(* IEC 61131-3 sources: eCockpitGit/test_project/src/%F%00 Library/%F%Common Functions/%F%Bits/%F%Bit Get Part, 8 files *)

(* ---- %POU%FU_bBitGetPart.st ---- *)
//This function gets only the needed bits of a variable
// |**Version**|**Author**| **Date** |**Changes**
// | 1         | NSN      | 16-03-22 | Creation
FUNCTION FU_bBitGetPart : BYTE
VAR_INPUT
	value			:BYTE;		//Variable to get value from
	amount			:BYTE;		//Amount of bits to change
	offset			:BYTE;		//Offset in variable to change bits at
END_VAR
(*%!%__DELIMITER__%!%*)
FU_bBitPartThrough		:=		SHR(value,offset) AND GConstants.binaryMaskByte[amount];

(* ---- %POU%FU_diBitGetPart.st ---- *)
//This function gets only the needed bits of a variable
// |**Version**|**Author**| **Date** |**Changes**
// | 1         | NSN      | 16-03-22 | Creation
FUNCTION FU_diBitGetPart : DINT
VAR_INPUT
	value			:DINT;		//Variable to get value from
	amount			:BYTE;		//Amount of bits to change
	offset			:BYTE;		//Offset in variable to change bits at
END_VAR
(*%!%__DELIMITER__%!%*)
FU_diBitGetPart		:=		TO_DINT(TO_UDINT(SHR(value,offset)) AND TO_UDINT(GConstants.binaryMaskDint[amount]));

(* ---- %POU%FU_dwBitGetPart.st ---- *)
//This function gets only the needed bits of a variable
// |**Version**|**Author**| **Date** |**Changes**
// | 1         | NSN      | 16-03-22 | Creation
FUNCTION FU_dwBitGetPart : DWORD
VAR_INPUT
	value			:DWORD;		//Variable to get value from
	amount			:BYTE;		//Amount of bits to change
	offset			:BYTE;		//Offset in variable to change bits at
END_VAR
(*%!%__DELIMITER__%!%*)
FU_dwBitGetPart		:=		SHR(value,offset) AND GConstants.binaryMaskDWord[amount];

(* ---- %POU%FU_iBitGetPart.st ---- *)
//This function gets only the needed bits of a variable
// |**Version**|**Author**| **Date** |**Changes**
// | 1         | NSN      | 16-03-22 | Creation
FUNCTION FU_iBitGetPart : INT
VAR_INPUT
	value			:INT;		//Variable to get value from
	amount			:BYTE;		//Amount of bits to change
	offset			:BYTE;		//Offset in variable to change bits at
END_VAR
(*%!%__DELIMITER__%!%*)
FU_iBitGetPart		:=		TO_INT(SHR(TO_UINT(value),offset) AND TO_UINT(GConstants.binaryMaskInt[amount]));

(* ---- %POU%FU_liBitGetPart.st ---- *)
//This function gets only the needed bits of a variable
// |**Version**|**Author**| **Date** |**Changes**
// | 1         | NSN      | 16-03-22 | Creation
FUNCTION FU_liBitGetPart : LINT
VAR_INPUT
	value			:LINT;		//Variable to get value from
	amount			:BYTE;		//Amount of bits to change
	offset			:BYTE;		//Offset in variable to change bits at
END_VAR
(*%!%__DELIMITER__%!%*)
FU_liBitGetPart		:=		TO_LINT(SHR(TO_ULINT(value),offset) AND TO_ULINT(GConstants.binaryMaskLint[amount]));

(* ---- %POU%FU_lwBitGetPart.st ---- *)
//This function gets only the needed bits of a variable
// |**Version**|**Author**| **Date** |**Changes**
// | 1         | NSN      | 16-03-22 | Creation
FUNCTION FU_lwBitGetPart : LWORD
VAR_INPUT
	value			:LWORD;		//Variable to get value from
	amount			:BYTE;		//Amount of bits to change
	offset			:BYTE;		//Offset in variable to change bits at
END_VAR
(*%!%__DELIMITER__%!%*)
FU_lwBitGetPart		:=		SHR(value,offset) AND GConstants.binaryMaskLWord[amount];

(* ---- %POU%FU_siBitGetPart.st ---- *)
//This function gets only the needed bits of a variable
// |**Version**|**Author**| **Date** |**Changes**
// | 1         | NSN      | 16-03-22 | Creation
FUNCTION FU_siBitGetPart : SINT
VAR_INPUT
	value			:SINT;		//Variable to get value from
	amount			:BYTE;		//Amount of bits to change
	offset			:BYTE;		//Offset in variable to change bits at
END_VAR
(*%!%__DELIMITER__%!%*)
FU_siBitGetPart		:=		TO_SINT(SHR(TO_USINT(value),offset) AND TO_USINT(GConstants.binaryMaskSint[amount]));

(* ---- %POU%FU_wBitGetPart.st ---- *)
//This function gets only the needed bits of a variable
// |**Version**|**Author**| **Date** |**Changes**
// | 1         | NSN      | 16-03-22 | Creation
FUNCTION FU_wBitGetPart : WORD
VAR_INPUT
	value			:WORD;		//Variable to get value from
	amount			:BYTE;		//Amount of bits to change
	offset			:BYTE;		//Offset in variable to change bits at
END_VAR
(*%!%__DELIMITER__%!%*)
FU_wBitGetPart		:=		SHR(value,offset) AND GConstants.binaryMaskWord[amount];
